PROGRAM MAIN
VAR
	fbModule1:	FB_Module01;
	fbComponent:	FB_ComponentEX;
END_VAR

fbModule1.M_Cycle();
fbComponent.M_Cycle();

END_PROGRAM

(* stored: Version 1.1.0.1
   POU MAIN: Id {2d4d4998-19ee-0f89-2021-34d743efb262}, SpecialFunc None *)
